FUNCTION_BLOCK InputPortCollection IMPLEMENTS I_InputPortCollection
VAR
	ports : Stack;
END_VAR

METHOD PUBLIC GetEnumerator : I_ForwardEnumerator
VAR_INPUT
END_VAR
GetEnumerator := ports.GetEnumerator();
END_METHOD

METHOD PUBLIC Insert
VAR_INPUT
	PortToInsert : I_InputPort;
END_VAR
ports.Push(PortToInsert);
END_METHOD

METHOD PUBLIC TryGetByName : BOOL;
VAR_INPUT
	Name : STRING;
	Destination : REFERENCE TO I_InputPort;
END_VAR
VAR
	portEnumerator : I_ForwardEnumerator;
	port : I_InputPort;
END_VAR
portEnumerator := ports.GetEnumerator();

WHILE portEnumerator.MoveNext() DO 
	IF  NOT portEnumerator.TryGet(port) THEN
		CONTINUE;
	END_IF
	
	IF port.Name = Name THEN 
		TryGetByName := TRUE;
		Destination := port;
		EXIT;
	END_IF

END_WHILE

portEnumerator.Dispose();
END_METHOD

END_FUNCTION_BLOCK

(* stored: Version 1.1.0.1, ProductVersion 3.1.4024.12
   POU InputPortCollection: Id {698d979b-c4a2-0ea2-2b7c-b5e4d16c5571}, SpecialFunc None
   Method GetEnumerator: Id {95dac596-2837-0680-0665-a50e69d8e327}
   Method Insert: Id {cb630fe7-ec89-0f7f-1cf8-60ccd4f6914b}
   Method TryGetByName: Id {428b5b08-e0a6-0f29-0910-d89eb64fe796} *)
